INTERFACE IReadOnlyPointerDictionary EXTENDS IPointerCollection

METHOD ContainsKey : BOOL
VAR_INPUT
	key : PVOID;
END_VAR
END_METHOD

METHOD GetKeyByIndex : PVOID
VAR_INPUT
	index : DINT;
END_VAR
END_METHOD

METHOD GetValueByIndex : PVOID
VAR_INPUT
	index : DINT;
END_VAR
END_METHOD

METHOD GetValueByKey : PVOID
VAR_INPUT
	key : PVOID;
END_VAR
END_METHOD

{attribute 'OPC.UA.DA.Property' := '1'}
{attribute 'monitoring' := 'call'}
PROPERTY KeyType : POINTER_TYPE
GET
END_GET
END_PROPERTY

{attribute 'OPC.UA.DA.Property' := '1'}
{attribute 'monitoring' := 'call'}
PROPERTY ValueType : POINTER_TYPE
GET
END_GET
END_PROPERTY

END_INTERFACE

(* stored: Version 1.1.0.1
   Itf IReadOnlyPointerDictionary: Id {2908c77a-1363-0667-2c19-5d19649147d8}
   Method ContainsKey: Id {790f9463-ea24-0924-136f-5261abf02f21}
   Method GetKeyByIndex: Id {5c886fa1-0056-01fe-220b-f37202feae98}
   Method GetValueByIndex: Id {2f02ddfc-52f6-0c61-0e1a-3b7b00d84670}
   Method GetValueByKey: Id {74202475-eeaa-034b-20ab-b4d0b23edae5}
   Property KeyType: Id {59ffd151-b89f-0c5d-0f9b-aac822ffded7}
   Get Get: Id {6746f417-f923-0481-0d78-ab2d32b071cb}
   Property ValueType: Id {9e7905ea-c2dc-011e-3d72-eb3aa8bc6729}
   Get Get: Id {4f6668d1-3920-010e-1057-e7c28fe98e5b} *)
